(* CoDeSys 2.3 export: GOLD.EXP *)

(* POU Mathematical/GOLD, ST *)
FUNCTION GOLD : REAL
VAR_INPUT
	X : REAL;
END_VAR


(*
version 1.1	10. mar. 2009
programmer 	hugo
tested by		tobias

this function calculates the golden function.

*)
GOLD := (X + SQRT(X*X + 4.0)) * 0.5;


(* revision history
hm	27. apr. 2008	rev 1.0
	original version

hm	10. mar. 2009	rev 1.1
	real constants updated to new systax using dot

*)
END_FUNCTION
